TYPE ST_PresetPosition :
STRUCT
    X : LREAL;
    Y : LREAL;
    Visited : BOOL;
END_STRUCT
END_TYPE

(* stored: Version 1.1.0.1, ProductVersion 3.1.4024.12
   DUT ST_PresetPosition: Id {ea251ab0-850c-4b87-b130-6620935d55ed} *)
